Universal Robots PolyScope program: recibir_str_socket.urp

Program recibir_str_socket (installation=default directory=/home/ur/ursim-current/programs createdIn=5.11.9.1010452 lastSavedIn=5.11.9.1010452 robotSerialNumber=20195699999)
Calibrated DH parameters: a=[0, -0.4784, -0.36, 0, 0, 0]; d=[0.1807, 0, 0, 0.17415, 0.11985, 0.11655]; alpha=[1.570796, 0, 0, 1.570796, -1.570796, 0]; deltaTheta=[0, 0, 0, 0, 0, 0]
BeforeStart
  conexion := False
  datos := [0,0,0,0]
  pos_pick := p[0,0,0,0,0,0]
Robot Program (runOnlyOnce=false)
  Loop While (checkContinuously=false) expression=conexion≟ False
    'Abrimos socket'
    conexion := socket_open("172.16.17.10",50000)
    Wait Sleep waitTime=0.01
  'Enviamos la cadena str "listo"'
  str := "listo"
  Script: socket_send_string(str)
  Loop While (checkContinuously=false) expression=datos[0]≠3
    'Leemos las tres comas flotantes'
    datos := socket_read_ascii_float(3)
    Wait Sleep waitTime=0.5
  'Guardamos las comas flotantes en variables'
  x := datos[1]
  y := datos[2]
  rz := datos[3]
  Script: socket_close()
  pos_pick := p[x,y,0,0,0,rz]
